PROGRAM MAIN
VAR
	i:UDINT;
	
END_VAR

//======FB Cyclic Update======

//模擬Index產生資料
FOR i:=0 TO GVL.Max_IndexNum-1 DO
	GVL.fbDataToNovRam[i]();
END_FOR

END_PROGRAM

(* stored: Version 1.1.0.1, ProductVersion 3.1.4024.11
   POU MAIN: Id {3ebd620b-e13f-4b0f-ae9c-4d4dc7ae0974}, SpecialFunc None *)
